{attribute 'global_init_slot' := '40500'}
VAR_GLOBAL
	Axis1_Prox AT %I* : BOOL;
	Axis2_Prox AT %I* : BOOL;
	Axis3_Prox AT %I* : BOOL;
	Axis4_Prox AT %I* : BOOL;
END_VAR

(* stored: Version 1.1.0.1, ProductVersion 3.1.4026.11
   GVL GVL_SteppersProx: Id {5b1115cf-ca8b-4b95-9e3f-ba6864fa250e} *)
